// TIA Portal V20 export
FUNCTION "SafetyState" : Void   // FC97, LAD
// stored: SetENOAutomatically false
   VAR CONSTANT
      TRUE : Bool := TRUE;
      FALSE : Bool;
   END_VAR
   VAR_TEMP   // added for the SCL form of the ladder/FBD networks
      _w1 : Bool;
   END_VAR
BEGIN

REGION Network 1: Stack Door Common Monitoring#1
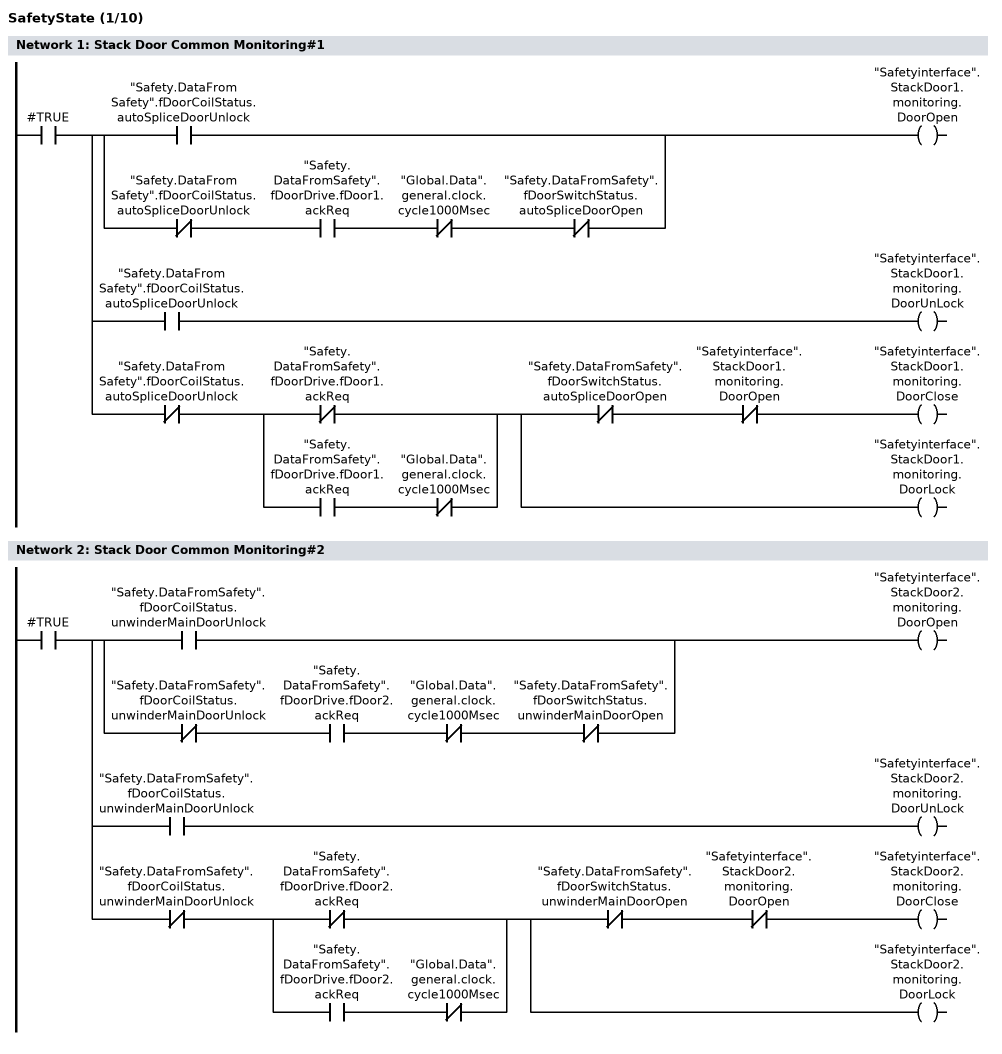
   RUNG wire#powerrail
      Contact( #TRUE )
      wire#w1
      Contact( "Safety.DataFromSafety".fDoorCoilStatus.autoSpliceDoorUnlock )
      wire#w2
      Coil( "Safetyinterface".StackDoor1.monitoring.DoorOpen )
   END_RUNG
   RUNG wire#w1
      I_Contact( "Safety.DataFromSafety".fDoorCoilStatus.autoSpliceDoorUnlock )
      Contact( "Safety.DataFromSafety".fDoorDrive.fDoor1.ackReq )
      I_Contact( "Global.Data".general.clock.cycle1000Msec )
      I_Contact( "Safety.DataFromSafety".fDoorSwitchStatus.autoSpliceDoorOpen )
   END_RUNG wire#w2
   RUNG wire#w1
      Contact( "Safety.DataFromSafety".fDoorCoilStatus.autoSpliceDoorUnlock )
      Coil( "Safetyinterface".StackDoor1.monitoring.DoorUnLock )
   END_RUNG
   RUNG wire#w1
      I_Contact( "Safety.DataFromSafety".fDoorCoilStatus.autoSpliceDoorUnlock )
      wire#w3
      I_Contact( "Safety.DataFromSafety".fDoorDrive.fDoor1.ackReq )
      wire#w4
      I_Contact( "Safety.DataFromSafety".fDoorSwitchStatus.autoSpliceDoorOpen )
      I_Contact( "Safetyinterface".StackDoor1.monitoring.DoorOpen )
      Coil( "Safetyinterface".StackDoor1.monitoring.DoorClose )
   END_RUNG
   RUNG wire#w3
      Contact( "Safety.DataFromSafety".fDoorDrive.fDoor1.ackReq )
      I_Contact( "Global.Data".general.clock.cycle1000Msec )
   END_RUNG wire#w4
   RUNG wire#w4
      Coil( "Safetyinterface".StackDoor1.monitoring.DoorLock )
   END_RUNG
   // the same network as SCL:
   "Safetyinterface".StackDoor1.monitoring.DoorOpen := #TRUE AND ("Safety.DataFromSafety".fDoorCoilStatus.autoSpliceDoorUnlock OR (NOT "Safety.DataFromSafety".fDoorCoilStatus.autoSpliceDoorUnlock AND "Safety.DataFromSafety".fDoorDrive.fDoor1.ackReq AND NOT "Global.Data".general.clock.cycle1000Msec AND NOT "Safety.DataFromSafety".fDoorSwitchStatus.autoSpliceDoorOpen));
   "Safetyinterface".StackDoor1.monitoring.DoorUnLock := #TRUE AND "Safety.DataFromSafety".fDoorCoilStatus.autoSpliceDoorUnlock;
   #_w1 := #TRUE AND NOT "Safety.DataFromSafety".fDoorCoilStatus.autoSpliceDoorUnlock AND (NOT "Safety.DataFromSafety".fDoorDrive.fDoor1.ackReq OR ("Safety.DataFromSafety".fDoorDrive.fDoor1.ackReq AND NOT "Global.Data".general.clock.cycle1000Msec));
   "Safetyinterface".StackDoor1.monitoring.DoorClose := #_w1 AND NOT "Safety.DataFromSafety".fDoorSwitchStatus.autoSpliceDoorOpen AND NOT "Safetyinterface".StackDoor1.monitoring.DoorOpen;
   "Safetyinterface".StackDoor1.monitoring.DoorLock := #_w1;
END_REGION

REGION Network 2: Stack Door Common Monitoring#2
   RUNG wire#powerrail
      Contact( #TRUE )
      wire#w1
      Contact( "Safety.DataFromSafety".fDoorCoilStatus.unwinderMainDoorUnlock )
      wire#w2
      Coil( "Safetyinterface".StackDoor2.monitoring.DoorOpen )
   END_RUNG
   RUNG wire#w1
      I_Contact( "Safety.DataFromSafety".fDoorCoilStatus.unwinderMainDoorUnlock )
      Contact( "Safety.DataFromSafety".fDoorDrive.fDoor2.ackReq )
      I_Contact( "Global.Data".general.clock.cycle1000Msec )
      I_Contact( "Safety.DataFromSafety".fDoorSwitchStatus.unwinderMainDoorOpen )
   END_RUNG wire#w2
   RUNG wire#w1
      Contact( "Safety.DataFromSafety".fDoorCoilStatus.unwinderMainDoorUnlock )
      Coil( "Safetyinterface".StackDoor2.monitoring.DoorUnLock )
   END_RUNG
   RUNG wire#w1
      I_Contact( "Safety.DataFromSafety".fDoorCoilStatus.unwinderMainDoorUnlock )
      wire#w3
      I_Contact( "Safety.DataFromSafety".fDoorDrive.fDoor2.ackReq )
      wire#w4
      I_Contact( "Safety.DataFromSafety".fDoorSwitchStatus.unwinderMainDoorOpen )
      I_Contact( "Safetyinterface".StackDoor2.monitoring.DoorOpen )
      Coil( "Safetyinterface".StackDoor2.monitoring.DoorClose )
   END_RUNG
   RUNG wire#w3
      Contact( "Safety.DataFromSafety".fDoorDrive.fDoor2.ackReq )
      I_Contact( "Global.Data".general.clock.cycle1000Msec )
   END_RUNG wire#w4
   RUNG wire#w4
      Coil( "Safetyinterface".StackDoor2.monitoring.DoorLock )
   END_RUNG
   // the same network as SCL:
   "Safetyinterface".StackDoor2.monitoring.DoorOpen := #TRUE AND ("Safety.DataFromSafety".fDoorCoilStatus.unwinderMainDoorUnlock OR (NOT "Safety.DataFromSafety".fDoorCoilStatus.unwinderMainDoorUnlock AND "Safety.DataFromSafety".fDoorDrive.fDoor2.ackReq AND NOT "Global.Data".general.clock.cycle1000Msec AND NOT "Safety.DataFromSafety".fDoorSwitchStatus.unwinderMainDoorOpen));
   "Safetyinterface".StackDoor2.monitoring.DoorUnLock := #TRUE AND "Safety.DataFromSafety".fDoorCoilStatus.unwinderMainDoorUnlock;
   #_w1 := #TRUE AND NOT "Safety.DataFromSafety".fDoorCoilStatus.unwinderMainDoorUnlock AND (NOT "Safety.DataFromSafety".fDoorDrive.fDoor2.ackReq OR ("Safety.DataFromSafety".fDoorDrive.fDoor2.ackReq AND NOT "Global.Data".general.clock.cycle1000Msec));
   "Safetyinterface".StackDoor2.monitoring.DoorClose := #_w1 AND NOT "Safety.DataFromSafety".fDoorSwitchStatus.unwinderMainDoorOpen AND NOT "Safetyinterface".StackDoor2.monitoring.DoorOpen;
   "Safetyinterface".StackDoor2.monitoring.DoorLock := #_w1;
END_REGION

REGION Network 3: Stack Door Common Monitoring#3
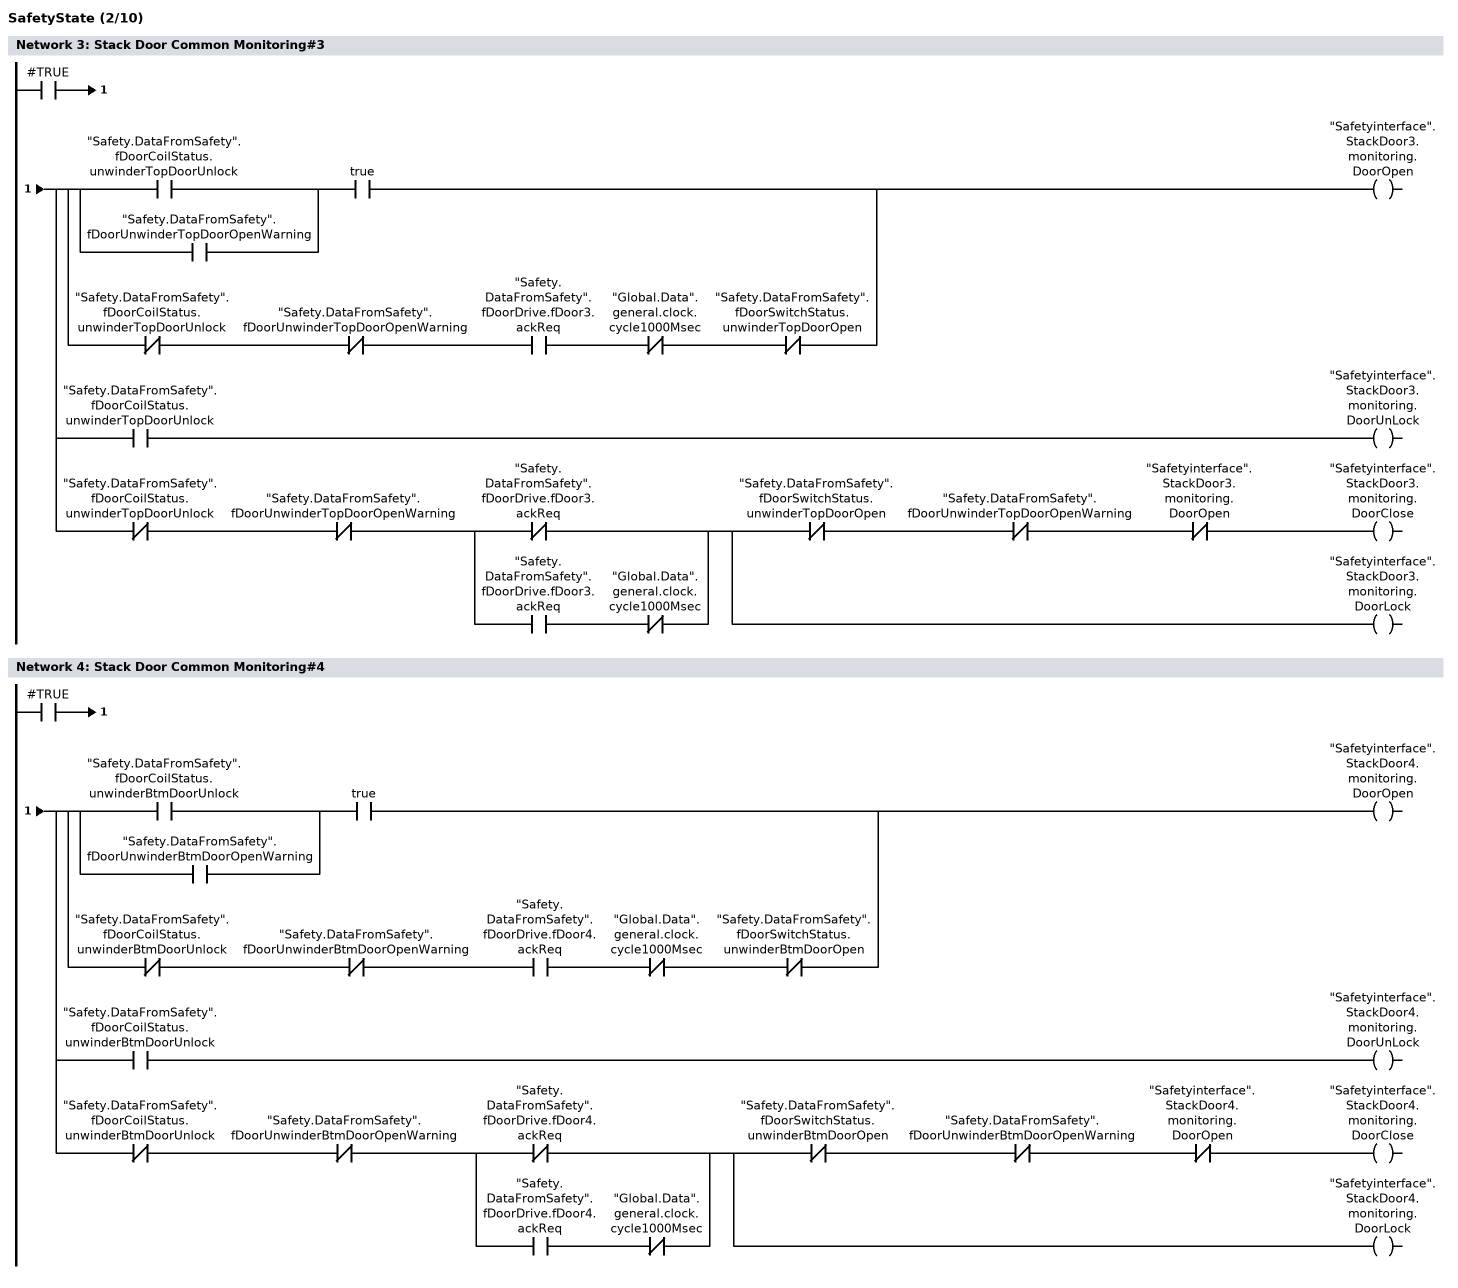
   RUNG wire#powerrail
      Contact( #TRUE )
      wire#w1
      Contact( "Safety.DataFromSafety".fDoorCoilStatus.unwinderTopDoorUnlock )
      wire#w2
      Contact( true )
      wire#w3
      Coil( "Safetyinterface".StackDoor3.monitoring.DoorOpen )
   END_RUNG
   RUNG wire#w1
      Contact( "Safety.DataFromSafety".fDoorUnwinderTopDoorOpenWarning )
   END_RUNG wire#w2
   RUNG wire#w1
      I_Contact( "Safety.DataFromSafety".fDoorCoilStatus.unwinderTopDoorUnlock )
      I_Contact( "Safety.DataFromSafety".fDoorUnwinderTopDoorOpenWarning )
      Contact( "Safety.DataFromSafety".fDoorDrive.fDoor3.ackReq )
      I_Contact( "Global.Data".general.clock.cycle1000Msec )
      I_Contact( "Safety.DataFromSafety".fDoorSwitchStatus.unwinderTopDoorOpen )
   END_RUNG wire#w3
   RUNG wire#w1
      Contact( "Safety.DataFromSafety".fDoorCoilStatus.unwinderTopDoorUnlock )
      Coil( "Safetyinterface".StackDoor3.monitoring.DoorUnLock )
   END_RUNG
   RUNG wire#w1
      I_Contact( "Safety.DataFromSafety".fDoorCoilStatus.unwinderTopDoorUnlock )
      I_Contact( "Safety.DataFromSafety".fDoorUnwinderTopDoorOpenWarning )
      wire#w4
      I_Contact( "Safety.DataFromSafety".fDoorDrive.fDoor3.ackReq )
      wire#w5
      I_Contact( "Safety.DataFromSafety".fDoorSwitchStatus.unwinderTopDoorOpen )
      I_Contact( "Safety.DataFromSafety".fDoorUnwinderTopDoorOpenWarning )
      I_Contact( "Safetyinterface".StackDoor3.monitoring.DoorOpen )
      Coil( "Safetyinterface".StackDoor3.monitoring.DoorClose )
   END_RUNG
   RUNG wire#w4
      Contact( "Safety.DataFromSafety".fDoorDrive.fDoor3.ackReq )
      I_Contact( "Global.Data".general.clock.cycle1000Msec )
   END_RUNG wire#w5
   RUNG wire#w5
      Coil( "Safetyinterface".StackDoor3.monitoring.DoorLock )
   END_RUNG
   // the same network as SCL:
   "Safetyinterface".StackDoor3.monitoring.DoorOpen := #TRUE AND ((("Safety.DataFromSafety".fDoorCoilStatus.unwinderTopDoorUnlock OR "Safety.DataFromSafety".fDoorUnwinderTopDoorOpenWarning) AND true) OR (NOT "Safety.DataFromSafety".fDoorCoilStatus.unwinderTopDoorUnlock AND NOT "Safety.DataFromSafety".fDoorUnwinderTopDoorOpenWarning AND "Safety.DataFromSafety".fDoorDrive.fDoor3.ackReq AND NOT "Global.Data".general.clock.cycle1000Msec AND NOT "Safety.DataFromSafety".fDoorSwitchStatus.unwinderTopDoorOpen));
   "Safetyinterface".StackDoor3.monitoring.DoorUnLock := #TRUE AND "Safety.DataFromSafety".fDoorCoilStatus.unwinderTopDoorUnlock;
   #_w1 := #TRUE AND NOT "Safety.DataFromSafety".fDoorCoilStatus.unwinderTopDoorUnlock AND NOT "Safety.DataFromSafety".fDoorUnwinderTopDoorOpenWarning AND (NOT "Safety.DataFromSafety".fDoorDrive.fDoor3.ackReq OR ("Safety.DataFromSafety".fDoorDrive.fDoor3.ackReq AND NOT "Global.Data".general.clock.cycle1000Msec));
   "Safetyinterface".StackDoor3.monitoring.DoorClose := #_w1 AND NOT "Safety.DataFromSafety".fDoorSwitchStatus.unwinderTopDoorOpen AND NOT "Safety.DataFromSafety".fDoorUnwinderTopDoorOpenWarning AND NOT "Safetyinterface".StackDoor3.monitoring.DoorOpen;
   "Safetyinterface".StackDoor3.monitoring.DoorLock := #_w1;
END_REGION

REGION Network 4: Stack Door Common Monitoring#4
   RUNG wire#powerrail
      Contact( #TRUE )
      wire#w1
      Contact( "Safety.DataFromSafety".fDoorCoilStatus.unwinderBtmDoorUnlock )
      wire#w2
      Contact( true )
      wire#w3
      Coil( "Safetyinterface".StackDoor4.monitoring.DoorOpen )
   END_RUNG
   RUNG wire#w1
      Contact( "Safety.DataFromSafety".fDoorUnwinderBtmDoorOpenWarning )
   END_RUNG wire#w2
   RUNG wire#w1
      I_Contact( "Safety.DataFromSafety".fDoorCoilStatus.unwinderBtmDoorUnlock )
      I_Contact( "Safety.DataFromSafety".fDoorUnwinderBtmDoorOpenWarning )
      Contact( "Safety.DataFromSafety".fDoorDrive.fDoor4.ackReq )
      I_Contact( "Global.Data".general.clock.cycle1000Msec )
      I_Contact( "Safety.DataFromSafety".fDoorSwitchStatus.unwinderBtmDoorOpen )
   END_RUNG wire#w3
   RUNG wire#w1
      Contact( "Safety.DataFromSafety".fDoorCoilStatus.unwinderBtmDoorUnlock )
      Coil( "Safetyinterface".StackDoor4.monitoring.DoorUnLock )
   END_RUNG
   RUNG wire#w1
      I_Contact( "Safety.DataFromSafety".fDoorCoilStatus.unwinderBtmDoorUnlock )
      I_Contact( "Safety.DataFromSafety".fDoorUnwinderBtmDoorOpenWarning )
      wire#w4
      I_Contact( "Safety.DataFromSafety".fDoorDrive.fDoor4.ackReq )
      wire#w5
      I_Contact( "Safety.DataFromSafety".fDoorSwitchStatus.unwinderBtmDoorOpen )
      I_Contact( "Safety.DataFromSafety".fDoorUnwinderBtmDoorOpenWarning )
      I_Contact( "Safetyinterface".StackDoor4.monitoring.DoorOpen )
      Coil( "Safetyinterface".StackDoor4.monitoring.DoorClose )
   END_RUNG
   RUNG wire#w4
      Contact( "Safety.DataFromSafety".fDoorDrive.fDoor4.ackReq )
      I_Contact( "Global.Data".general.clock.cycle1000Msec )
   END_RUNG wire#w5
   RUNG wire#w5
      Coil( "Safetyinterface".StackDoor4.monitoring.DoorLock )
   END_RUNG
   // the same network as SCL:
   "Safetyinterface".StackDoor4.monitoring.DoorOpen := #TRUE AND ((("Safety.DataFromSafety".fDoorCoilStatus.unwinderBtmDoorUnlock OR "Safety.DataFromSafety".fDoorUnwinderBtmDoorOpenWarning) AND true) OR (NOT "Safety.DataFromSafety".fDoorCoilStatus.unwinderBtmDoorUnlock AND NOT "Safety.DataFromSafety".fDoorUnwinderBtmDoorOpenWarning AND "Safety.DataFromSafety".fDoorDrive.fDoor4.ackReq AND NOT "Global.Data".general.clock.cycle1000Msec AND NOT "Safety.DataFromSafety".fDoorSwitchStatus.unwinderBtmDoorOpen));
   "Safetyinterface".StackDoor4.monitoring.DoorUnLock := #TRUE AND "Safety.DataFromSafety".fDoorCoilStatus.unwinderBtmDoorUnlock;
   #_w1 := #TRUE AND NOT "Safety.DataFromSafety".fDoorCoilStatus.unwinderBtmDoorUnlock AND NOT "Safety.DataFromSafety".fDoorUnwinderBtmDoorOpenWarning AND (NOT "Safety.DataFromSafety".fDoorDrive.fDoor4.ackReq OR ("Safety.DataFromSafety".fDoorDrive.fDoor4.ackReq AND NOT "Global.Data".general.clock.cycle1000Msec));
   "Safetyinterface".StackDoor4.monitoring.DoorClose := #_w1 AND NOT "Safety.DataFromSafety".fDoorSwitchStatus.unwinderBtmDoorOpen AND NOT "Safety.DataFromSafety".fDoorUnwinderBtmDoorOpenWarning AND NOT "Safetyinterface".StackDoor4.monitoring.DoorOpen;
   "Safetyinterface".StackDoor4.monitoring.DoorLock := #_w1;
END_REGION

REGION Network 5: Stack Door Common Command#5
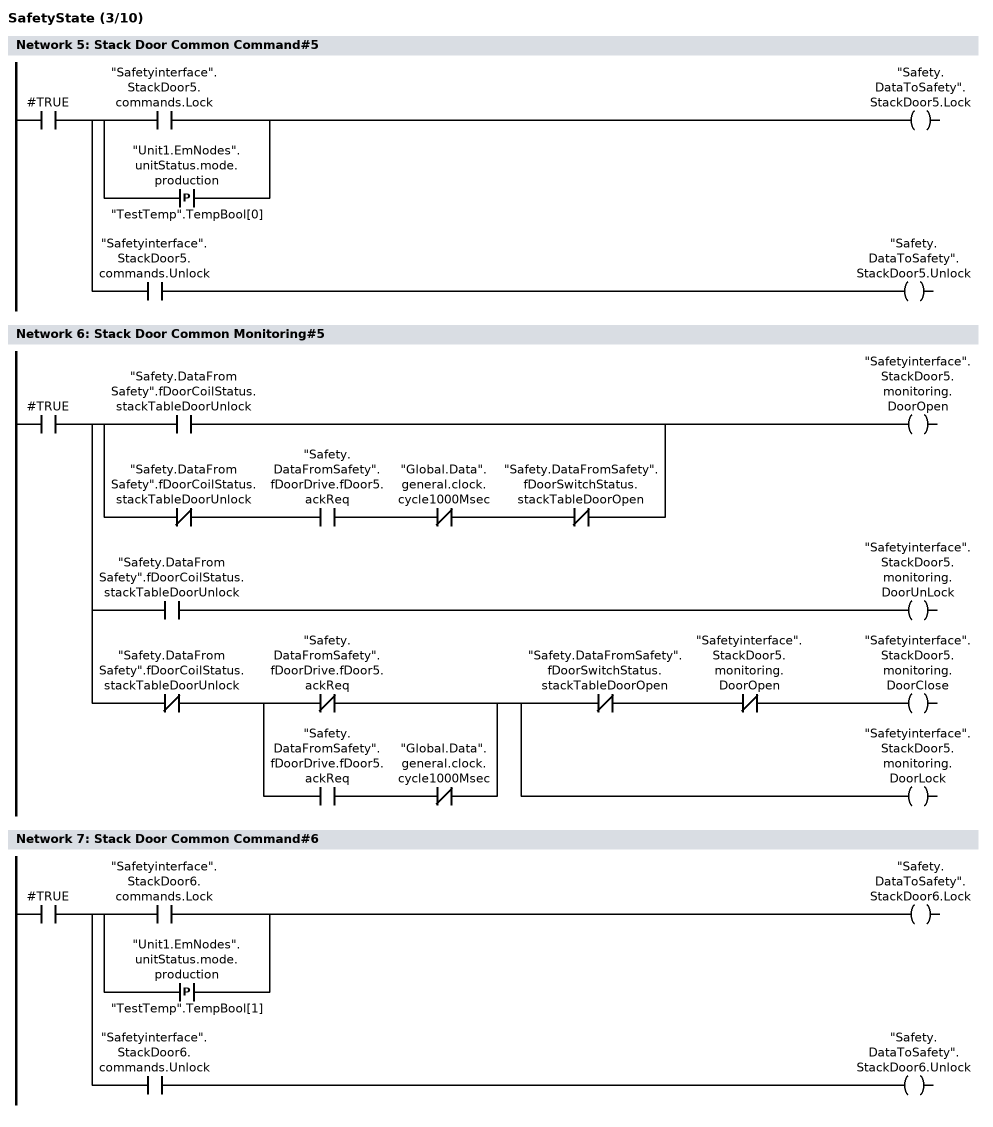
   RUNG wire#powerrail
      Contact( #TRUE )
      wire#w1
      Contact( "Safetyinterface".StackDoor5.commands.Lock )
      wire#w2
      Coil( "Safety.DataToSafety".StackDoor5.Lock )
   END_RUNG
   RUNG wire#w1
      P_Contact(operand := "Unit1.EmNodes".unitStatus.mode.production, bit := "TestTemp".TempBool[0])
   END_RUNG wire#w2
   RUNG wire#w1
      Contact( "Safetyinterface".StackDoor5.commands.Unlock )
      Coil( "Safety.DataToSafety".StackDoor5.Unlock )
   END_RUNG
   // the same network as SCL:
   #_w1 := #TRUE AND "Unit1.EmNodes".unitStatus.mode.production AND NOT "TestTemp".TempBool[0];   // rising edge of "Unit1.EmNodes".unitStatus.mode.production
   "TestTemp".TempBool[0] := "Unit1.EmNodes".unitStatus.mode.production;
   "Safety.DataToSafety".StackDoor5.Lock := (#TRUE AND "Safetyinterface".StackDoor5.commands.Lock) OR #_w1;
   "Safety.DataToSafety".StackDoor5.Unlock := #TRUE AND "Safetyinterface".StackDoor5.commands.Unlock;
END_REGION

REGION Network 6: Stack Door Common Monitoring#5
   RUNG wire#powerrail
      Contact( #TRUE )
      wire#w1
      Contact( "Safety.DataFromSafety".fDoorCoilStatus.stackTableDoorUnlock )
      wire#w2
      Coil( "Safetyinterface".StackDoor5.monitoring.DoorOpen )
   END_RUNG
   RUNG wire#w1
      I_Contact( "Safety.DataFromSafety".fDoorCoilStatus.stackTableDoorUnlock )
      Contact( "Safety.DataFromSafety".fDoorDrive.fDoor5.ackReq )
      I_Contact( "Global.Data".general.clock.cycle1000Msec )
      I_Contact( "Safety.DataFromSafety".fDoorSwitchStatus.stackTableDoorOpen )
   END_RUNG wire#w2
   RUNG wire#w1
      Contact( "Safety.DataFromSafety".fDoorCoilStatus.stackTableDoorUnlock )
      Coil( "Safetyinterface".StackDoor5.monitoring.DoorUnLock )
   END_RUNG
   RUNG wire#w1
      I_Contact( "Safety.DataFromSafety".fDoorCoilStatus.stackTableDoorUnlock )
      wire#w3
      I_Contact( "Safety.DataFromSafety".fDoorDrive.fDoor5.ackReq )
      wire#w4
      I_Contact( "Safety.DataFromSafety".fDoorSwitchStatus.stackTableDoorOpen )
      I_Contact( "Safetyinterface".StackDoor5.monitoring.DoorOpen )
      Coil( "Safetyinterface".StackDoor5.monitoring.DoorClose )
   END_RUNG
   RUNG wire#w3
      Contact( "Safety.DataFromSafety".fDoorDrive.fDoor5.ackReq )
      I_Contact( "Global.Data".general.clock.cycle1000Msec )
   END_RUNG wire#w4
   RUNG wire#w4
      Coil( "Safetyinterface".StackDoor5.monitoring.DoorLock )
   END_RUNG
   // the same network as SCL:
   "Safetyinterface".StackDoor5.monitoring.DoorOpen := #TRUE AND ("Safety.DataFromSafety".fDoorCoilStatus.stackTableDoorUnlock OR (NOT "Safety.DataFromSafety".fDoorCoilStatus.stackTableDoorUnlock AND "Safety.DataFromSafety".fDoorDrive.fDoor5.ackReq AND NOT "Global.Data".general.clock.cycle1000Msec AND NOT "Safety.DataFromSafety".fDoorSwitchStatus.stackTableDoorOpen));
   "Safetyinterface".StackDoor5.monitoring.DoorUnLock := #TRUE AND "Safety.DataFromSafety".fDoorCoilStatus.stackTableDoorUnlock;
   #_w1 := #TRUE AND NOT "Safety.DataFromSafety".fDoorCoilStatus.stackTableDoorUnlock AND (NOT "Safety.DataFromSafety".fDoorDrive.fDoor5.ackReq OR ("Safety.DataFromSafety".fDoorDrive.fDoor5.ackReq AND NOT "Global.Data".general.clock.cycle1000Msec));
   "Safetyinterface".StackDoor5.monitoring.DoorClose := #_w1 AND NOT "Safety.DataFromSafety".fDoorSwitchStatus.stackTableDoorOpen AND NOT "Safetyinterface".StackDoor5.monitoring.DoorOpen;
   "Safetyinterface".StackDoor5.monitoring.DoorLock := #_w1;
END_REGION

REGION Network 7: Stack Door Common Command#6
   RUNG wire#powerrail
      Contact( #TRUE )
      wire#w1
      Contact( "Safetyinterface".StackDoor6.commands.Lock )
      wire#w2
      Coil( "Safety.DataToSafety".StackDoor6.Lock )
   END_RUNG
   RUNG wire#w1
      P_Contact(operand := "Unit1.EmNodes".unitStatus.mode.production, bit := "TestTemp".TempBool[1])
   END_RUNG wire#w2
   RUNG wire#w1
      Contact( "Safetyinterface".StackDoor6.commands.Unlock )
      Coil( "Safety.DataToSafety".StackDoor6.Unlock )
   END_RUNG
   // the same network as SCL:
   #_w1 := #TRUE AND "Unit1.EmNodes".unitStatus.mode.production AND NOT "TestTemp".TempBool[1];   // rising edge of "Unit1.EmNodes".unitStatus.mode.production
   "TestTemp".TempBool[1] := "Unit1.EmNodes".unitStatus.mode.production;
   "Safety.DataToSafety".StackDoor6.Lock := (#TRUE AND "Safetyinterface".StackDoor6.commands.Lock) OR #_w1;
   "Safety.DataToSafety".StackDoor6.Unlock := #TRUE AND "Safetyinterface".StackDoor6.commands.Unlock;
END_REGION

REGION Network 8: Stack Door Common Monitoring#6
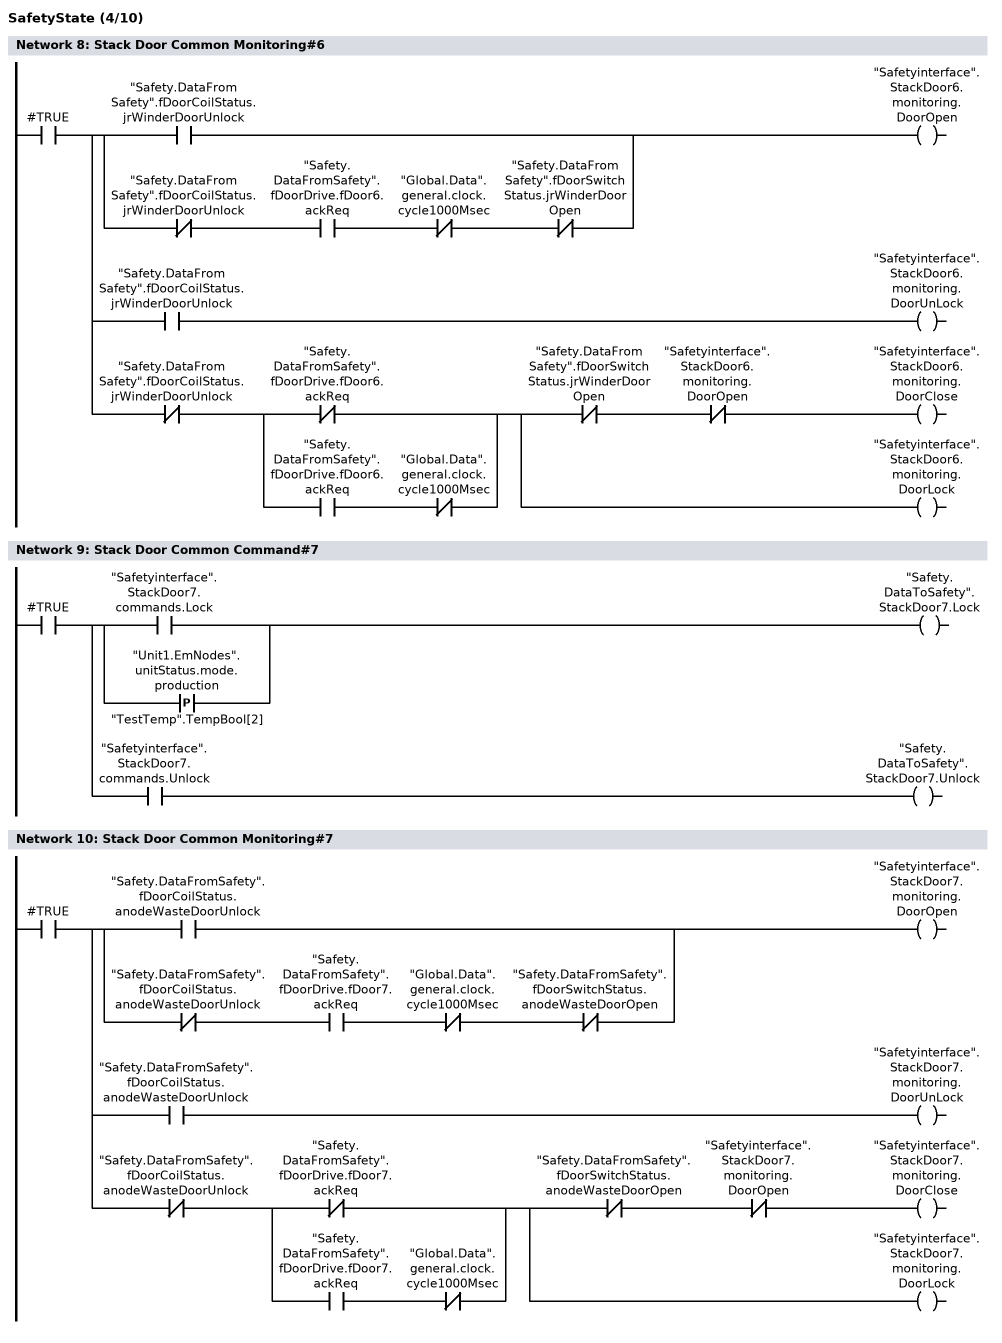
   RUNG wire#powerrail
      Contact( #TRUE )
      wire#w1
      Contact( "Safety.DataFromSafety".fDoorCoilStatus.jrWinderDoorUnlock )
      wire#w2
      Coil( "Safetyinterface".StackDoor6.monitoring.DoorOpen )
   END_RUNG
   RUNG wire#w1
      I_Contact( "Safety.DataFromSafety".fDoorCoilStatus.jrWinderDoorUnlock )
      Contact( "Safety.DataFromSafety".fDoorDrive.fDoor6.ackReq )
      I_Contact( "Global.Data".general.clock.cycle1000Msec )
      I_Contact( "Safety.DataFromSafety".fDoorSwitchStatus.jrWinderDoorOpen )
   END_RUNG wire#w2
   RUNG wire#w1
      Contact( "Safety.DataFromSafety".fDoorCoilStatus.jrWinderDoorUnlock )
      Coil( "Safetyinterface".StackDoor6.monitoring.DoorUnLock )
   END_RUNG
   RUNG wire#w1
      I_Contact( "Safety.DataFromSafety".fDoorCoilStatus.jrWinderDoorUnlock )
      wire#w3
      I_Contact( "Safety.DataFromSafety".fDoorDrive.fDoor6.ackReq )
      wire#w4
      I_Contact( "Safety.DataFromSafety".fDoorSwitchStatus.jrWinderDoorOpen )
      I_Contact( "Safetyinterface".StackDoor6.monitoring.DoorOpen )
      Coil( "Safetyinterface".StackDoor6.monitoring.DoorClose )
   END_RUNG
   RUNG wire#w3
      Contact( "Safety.DataFromSafety".fDoorDrive.fDoor6.ackReq )
      I_Contact( "Global.Data".general.clock.cycle1000Msec )
   END_RUNG wire#w4
   RUNG wire#w4
      Coil( "Safetyinterface".StackDoor6.monitoring.DoorLock )
   END_RUNG
   // the same network as SCL:
   "Safetyinterface".StackDoor6.monitoring.DoorOpen := #TRUE AND ("Safety.DataFromSafety".fDoorCoilStatus.jrWinderDoorUnlock OR (NOT "Safety.DataFromSafety".fDoorCoilStatus.jrWinderDoorUnlock AND "Safety.DataFromSafety".fDoorDrive.fDoor6.ackReq AND NOT "Global.Data".general.clock.cycle1000Msec AND NOT "Safety.DataFromSafety".fDoorSwitchStatus.jrWinderDoorOpen));
   "Safetyinterface".StackDoor6.monitoring.DoorUnLock := #TRUE AND "Safety.DataFromSafety".fDoorCoilStatus.jrWinderDoorUnlock;
   #_w1 := #TRUE AND NOT "Safety.DataFromSafety".fDoorCoilStatus.jrWinderDoorUnlock AND (NOT "Safety.DataFromSafety".fDoorDrive.fDoor6.ackReq OR ("Safety.DataFromSafety".fDoorDrive.fDoor6.ackReq AND NOT "Global.Data".general.clock.cycle1000Msec));
   "Safetyinterface".StackDoor6.monitoring.DoorClose := #_w1 AND NOT "Safety.DataFromSafety".fDoorSwitchStatus.jrWinderDoorOpen AND NOT "Safetyinterface".StackDoor6.monitoring.DoorOpen;
   "Safetyinterface".StackDoor6.monitoring.DoorLock := #_w1;
END_REGION

REGION Network 9: Stack Door Common Command#7
   RUNG wire#powerrail
      Contact( #TRUE )
      wire#w1
      Contact( "Safetyinterface".StackDoor7.commands.Lock )
      wire#w2
      Coil( "Safety.DataToSafety".StackDoor7.Lock )
   END_RUNG
   RUNG wire#w1
      P_Contact(operand := "Unit1.EmNodes".unitStatus.mode.production, bit := "TestTemp".TempBool[2])
   END_RUNG wire#w2
   RUNG wire#w1
      Contact( "Safetyinterface".StackDoor7.commands.Unlock )
      Coil( "Safety.DataToSafety".StackDoor7.Unlock )
   END_RUNG
   // the same network as SCL:
   #_w1 := #TRUE AND "Unit1.EmNodes".unitStatus.mode.production AND NOT "TestTemp".TempBool[2];   // rising edge of "Unit1.EmNodes".unitStatus.mode.production
   "TestTemp".TempBool[2] := "Unit1.EmNodes".unitStatus.mode.production;
   "Safety.DataToSafety".StackDoor7.Lock := (#TRUE AND "Safetyinterface".StackDoor7.commands.Lock) OR #_w1;
   "Safety.DataToSafety".StackDoor7.Unlock := #TRUE AND "Safetyinterface".StackDoor7.commands.Unlock;
END_REGION

REGION Network 10: Stack Door Common Monitoring#7
   RUNG wire#powerrail
      Contact( #TRUE )
      wire#w1
      Contact( "Safety.DataFromSafety".fDoorCoilStatus.anodeWasteDoorUnlock )
      wire#w2
      Coil( "Safetyinterface".StackDoor7.monitoring.DoorOpen )
   END_RUNG
   RUNG wire#w1
      I_Contact( "Safety.DataFromSafety".fDoorCoilStatus.anodeWasteDoorUnlock )
      Contact( "Safety.DataFromSafety".fDoorDrive.fDoor7.ackReq )
      I_Contact( "Global.Data".general.clock.cycle1000Msec )
      I_Contact( "Safety.DataFromSafety".fDoorSwitchStatus.anodeWasteDoorOpen )
   END_RUNG wire#w2
   RUNG wire#w1
      Contact( "Safety.DataFromSafety".fDoorCoilStatus.anodeWasteDoorUnlock )
      Coil( "Safetyinterface".StackDoor7.monitoring.DoorUnLock )
   END_RUNG
   RUNG wire#w1
      I_Contact( "Safety.DataFromSafety".fDoorCoilStatus.anodeWasteDoorUnlock )
      wire#w3
      I_Contact( "Safety.DataFromSafety".fDoorDrive.fDoor7.ackReq )
      wire#w4
      I_Contact( "Safety.DataFromSafety".fDoorSwitchStatus.anodeWasteDoorOpen )
      I_Contact( "Safetyinterface".StackDoor7.monitoring.DoorOpen )
      Coil( "Safetyinterface".StackDoor7.monitoring.DoorClose )
   END_RUNG
   RUNG wire#w3
      Contact( "Safety.DataFromSafety".fDoorDrive.fDoor7.ackReq )
      I_Contact( "Global.Data".general.clock.cycle1000Msec )
   END_RUNG wire#w4
   RUNG wire#w4
      Coil( "Safetyinterface".StackDoor7.monitoring.DoorLock )
   END_RUNG
   // the same network as SCL:
   "Safetyinterface".StackDoor7.monitoring.DoorOpen := #TRUE AND ("Safety.DataFromSafety".fDoorCoilStatus.anodeWasteDoorUnlock OR (NOT "Safety.DataFromSafety".fDoorCoilStatus.anodeWasteDoorUnlock AND "Safety.DataFromSafety".fDoorDrive.fDoor7.ackReq AND NOT "Global.Data".general.clock.cycle1000Msec AND NOT "Safety.DataFromSafety".fDoorSwitchStatus.anodeWasteDoorOpen));
   "Safetyinterface".StackDoor7.monitoring.DoorUnLock := #TRUE AND "Safety.DataFromSafety".fDoorCoilStatus.anodeWasteDoorUnlock;
   #_w1 := #TRUE AND NOT "Safety.DataFromSafety".fDoorCoilStatus.anodeWasteDoorUnlock AND (NOT "Safety.DataFromSafety".fDoorDrive.fDoor7.ackReq OR ("Safety.DataFromSafety".fDoorDrive.fDoor7.ackReq AND NOT "Global.Data".general.clock.cycle1000Msec));
   "Safetyinterface".StackDoor7.monitoring.DoorClose := #_w1 AND NOT "Safety.DataFromSafety".fDoorSwitchStatus.anodeWasteDoorOpen AND NOT "Safetyinterface".StackDoor7.monitoring.DoorOpen;
   "Safetyinterface".StackDoor7.monitoring.DoorLock := #_w1;
END_REGION

REGION Network 11: Stack Door Common Command#8
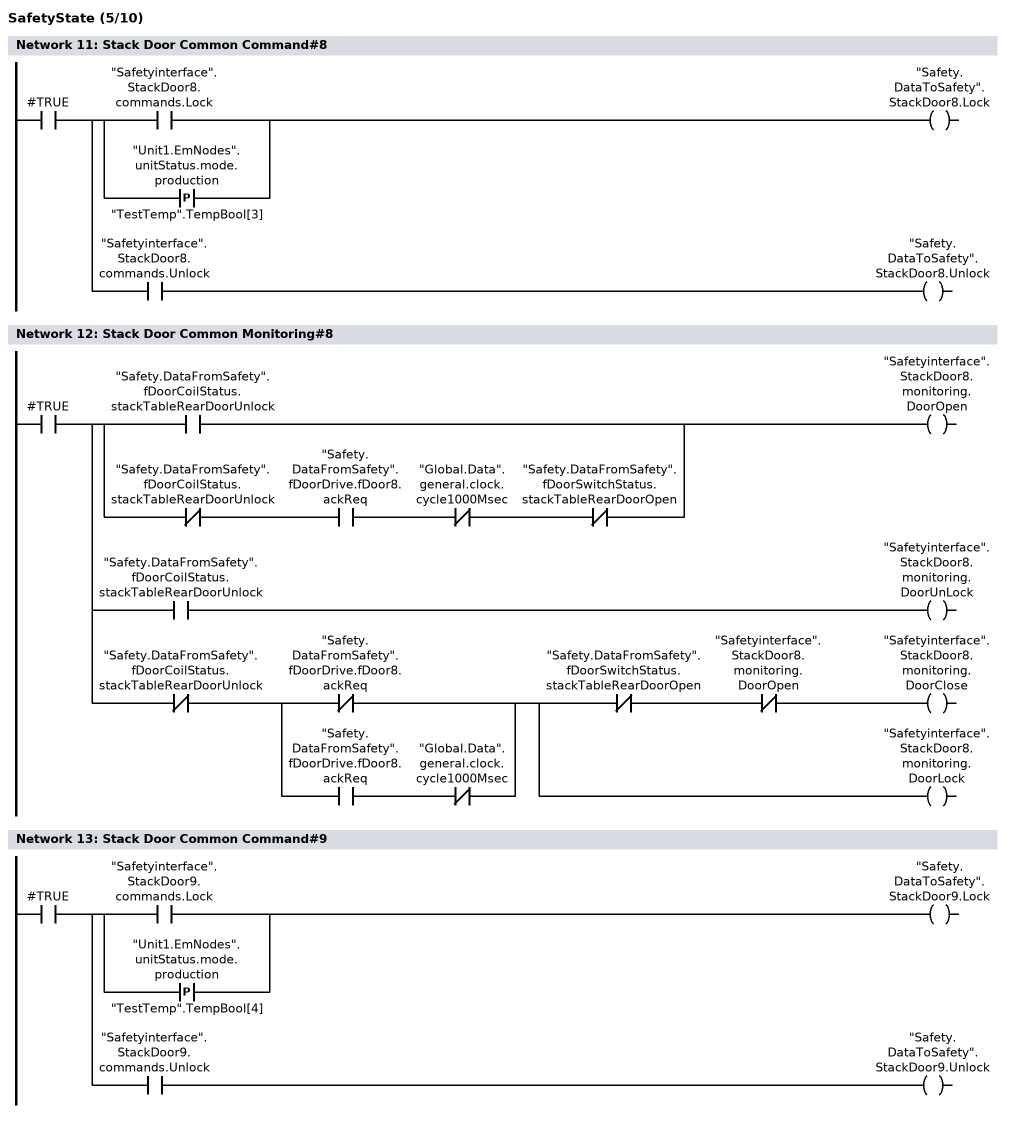
   RUNG wire#powerrail
      Contact( #TRUE )
      wire#w1
      Contact( "Safetyinterface".StackDoor8.commands.Lock )
      wire#w2
      Coil( "Safety.DataToSafety".StackDoor8.Lock )
   END_RUNG
   RUNG wire#w1
      P_Contact(operand := "Unit1.EmNodes".unitStatus.mode.production, bit := "TestTemp".TempBool[3])
   END_RUNG wire#w2
   RUNG wire#w1
      Contact( "Safetyinterface".StackDoor8.commands.Unlock )
      Coil( "Safety.DataToSafety".StackDoor8.Unlock )
   END_RUNG
   // the same network as SCL:
   #_w1 := #TRUE AND "Unit1.EmNodes".unitStatus.mode.production AND NOT "TestTemp".TempBool[3];   // rising edge of "Unit1.EmNodes".unitStatus.mode.production
   "TestTemp".TempBool[3] := "Unit1.EmNodes".unitStatus.mode.production;
   "Safety.DataToSafety".StackDoor8.Lock := (#TRUE AND "Safetyinterface".StackDoor8.commands.Lock) OR #_w1;
   "Safety.DataToSafety".StackDoor8.Unlock := #TRUE AND "Safetyinterface".StackDoor8.commands.Unlock;
END_REGION

REGION Network 12: Stack Door Common Monitoring#8
   RUNG wire#powerrail
      Contact( #TRUE )
      wire#w1
      Contact( "Safety.DataFromSafety".fDoorCoilStatus.stackTableRearDoorUnlock )
      wire#w2
      Coil( "Safetyinterface".StackDoor8.monitoring.DoorOpen )
   END_RUNG
   RUNG wire#w1
      I_Contact( "Safety.DataFromSafety".fDoorCoilStatus.stackTableRearDoorUnlock )
      Contact( "Safety.DataFromSafety".fDoorDrive.fDoor8.ackReq )
      I_Contact( "Global.Data".general.clock.cycle1000Msec )
      I_Contact( "Safety.DataFromSafety".fDoorSwitchStatus.stackTableRearDoorOpen )
   END_RUNG wire#w2
   RUNG wire#w1
      Contact( "Safety.DataFromSafety".fDoorCoilStatus.stackTableRearDoorUnlock )
      Coil( "Safetyinterface".StackDoor8.monitoring.DoorUnLock )
   END_RUNG
   RUNG wire#w1
      I_Contact( "Safety.DataFromSafety".fDoorCoilStatus.stackTableRearDoorUnlock )
      wire#w3
      I_Contact( "Safety.DataFromSafety".fDoorDrive.fDoor8.ackReq )
      wire#w4
      I_Contact( "Safety.DataFromSafety".fDoorSwitchStatus.stackTableRearDoorOpen )
      I_Contact( "Safetyinterface".StackDoor8.monitoring.DoorOpen )
      Coil( "Safetyinterface".StackDoor8.monitoring.DoorClose )
   END_RUNG
   RUNG wire#w3
      Contact( "Safety.DataFromSafety".fDoorDrive.fDoor8.ackReq )
      I_Contact( "Global.Data".general.clock.cycle1000Msec )
   END_RUNG wire#w4
   RUNG wire#w4
      Coil( "Safetyinterface".StackDoor8.monitoring.DoorLock )
   END_RUNG
   // the same network as SCL:
   "Safetyinterface".StackDoor8.monitoring.DoorOpen := #TRUE AND ("Safety.DataFromSafety".fDoorCoilStatus.stackTableRearDoorUnlock OR (NOT "Safety.DataFromSafety".fDoorCoilStatus.stackTableRearDoorUnlock AND "Safety.DataFromSafety".fDoorDrive.fDoor8.ackReq AND NOT "Global.Data".general.clock.cycle1000Msec AND NOT "Safety.DataFromSafety".fDoorSwitchStatus.stackTableRearDoorOpen));
   "Safetyinterface".StackDoor8.monitoring.DoorUnLock := #TRUE AND "Safety.DataFromSafety".fDoorCoilStatus.stackTableRearDoorUnlock;
   #_w1 := #TRUE AND NOT "Safety.DataFromSafety".fDoorCoilStatus.stackTableRearDoorUnlock AND (NOT "Safety.DataFromSafety".fDoorDrive.fDoor8.ackReq OR ("Safety.DataFromSafety".fDoorDrive.fDoor8.ackReq AND NOT "Global.Data".general.clock.cycle1000Msec));
   "Safetyinterface".StackDoor8.monitoring.DoorClose := #_w1 AND NOT "Safety.DataFromSafety".fDoorSwitchStatus.stackTableRearDoorOpen AND NOT "Safetyinterface".StackDoor8.monitoring.DoorOpen;
   "Safetyinterface".StackDoor8.monitoring.DoorLock := #_w1;
END_REGION

REGION Network 13: Stack Door Common Command#9
   RUNG wire#powerrail
      Contact( #TRUE )
      wire#w1
      Contact( "Safetyinterface".StackDoor9.commands.Lock )
      wire#w2
      Coil( "Safety.DataToSafety".StackDoor9.Lock )
   END_RUNG
   RUNG wire#w1
      P_Contact(operand := "Unit1.EmNodes".unitStatus.mode.production, bit := "TestTemp".TempBool[4])
   END_RUNG wire#w2
   RUNG wire#w1
      Contact( "Safetyinterface".StackDoor9.commands.Unlock )
      Coil( "Safety.DataToSafety".StackDoor9.Unlock )
   END_RUNG
   // the same network as SCL:
   #_w1 := #TRUE AND "Unit1.EmNodes".unitStatus.mode.production AND NOT "TestTemp".TempBool[4];   // rising edge of "Unit1.EmNodes".unitStatus.mode.production
   "TestTemp".TempBool[4] := "Unit1.EmNodes".unitStatus.mode.production;
   "Safety.DataToSafety".StackDoor9.Lock := (#TRUE AND "Safetyinterface".StackDoor9.commands.Lock) OR #_w1;
   "Safety.DataToSafety".StackDoor9.Unlock := #TRUE AND "Safetyinterface".StackDoor9.commands.Unlock;
END_REGION

REGION Network 14: Stack Door Common Monitoring#9
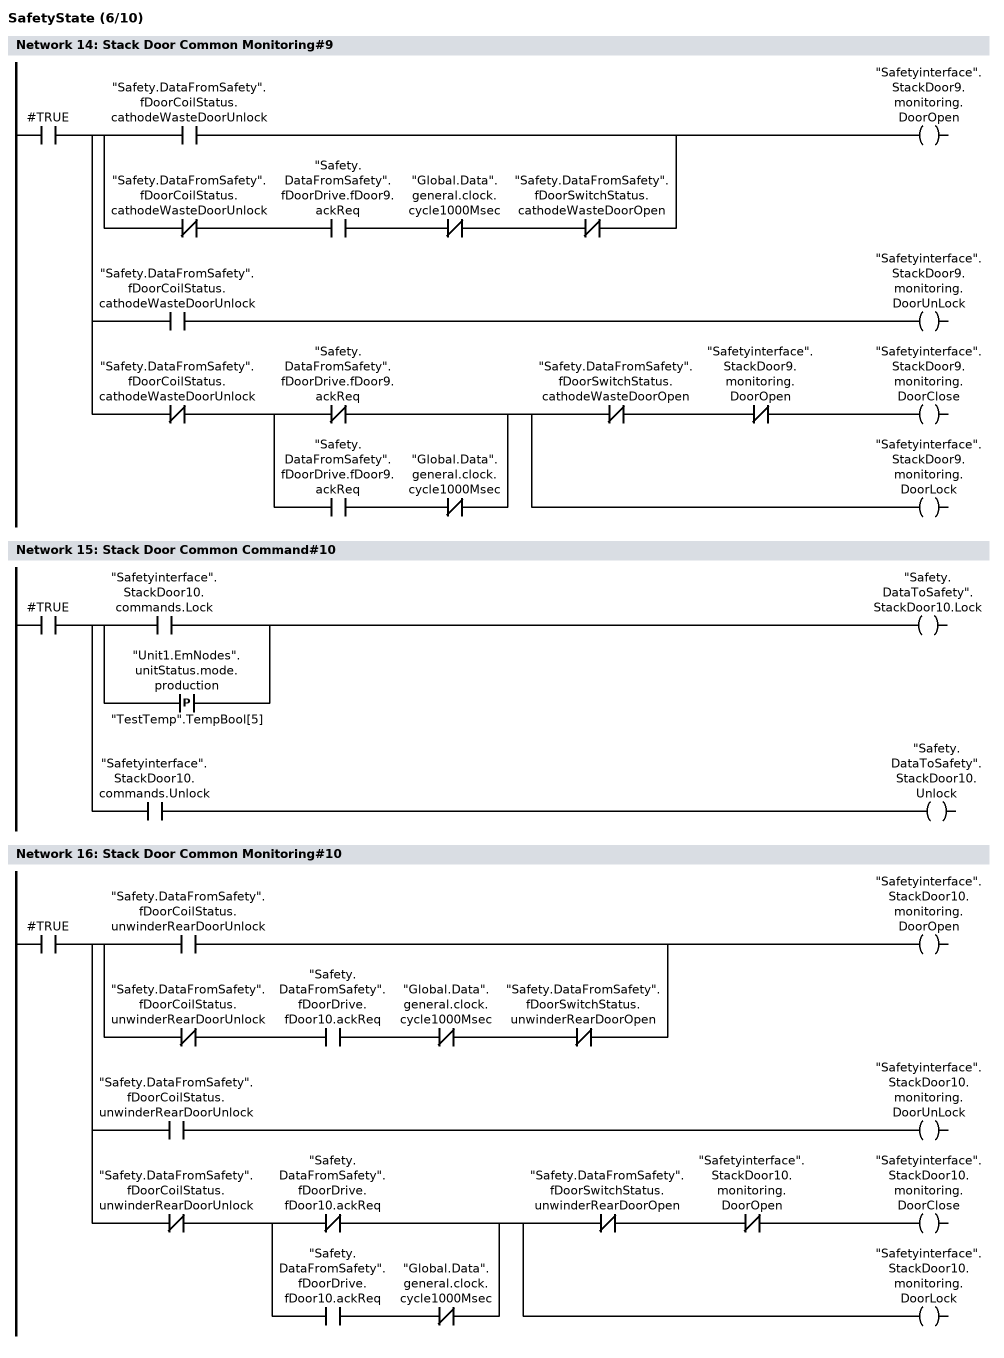
   RUNG wire#powerrail
      Contact( #TRUE )
      wire#w1
      Contact( "Safety.DataFromSafety".fDoorCoilStatus.cathodeWasteDoorUnlock )
      wire#w2
      Coil( "Safetyinterface".StackDoor9.monitoring.DoorOpen )
   END_RUNG
   RUNG wire#w1
      I_Contact( "Safety.DataFromSafety".fDoorCoilStatus.cathodeWasteDoorUnlock )
      Contact( "Safety.DataFromSafety".fDoorDrive.fDoor9.ackReq )
      I_Contact( "Global.Data".general.clock.cycle1000Msec )
      I_Contact( "Safety.DataFromSafety".fDoorSwitchStatus.cathodeWasteDoorOpen )
   END_RUNG wire#w2
   RUNG wire#w1
      Contact( "Safety.DataFromSafety".fDoorCoilStatus.cathodeWasteDoorUnlock )
      Coil( "Safetyinterface".StackDoor9.monitoring.DoorUnLock )
   END_RUNG
   RUNG wire#w1
      I_Contact( "Safety.DataFromSafety".fDoorCoilStatus.cathodeWasteDoorUnlock )
      wire#w3
      I_Contact( "Safety.DataFromSafety".fDoorDrive.fDoor9.ackReq )
      wire#w4
      I_Contact( "Safety.DataFromSafety".fDoorSwitchStatus.cathodeWasteDoorOpen )
      I_Contact( "Safetyinterface".StackDoor9.monitoring.DoorOpen )
      Coil( "Safetyinterface".StackDoor9.monitoring.DoorClose )
   END_RUNG
   RUNG wire#w3
      Contact( "Safety.DataFromSafety".fDoorDrive.fDoor9.ackReq )
      I_Contact( "Global.Data".general.clock.cycle1000Msec )
   END_RUNG wire#w4
   RUNG wire#w4
      Coil( "Safetyinterface".StackDoor9.monitoring.DoorLock )
   END_RUNG
   // the same network as SCL:
   "Safetyinterface".StackDoor9.monitoring.DoorOpen := #TRUE AND ("Safety.DataFromSafety".fDoorCoilStatus.cathodeWasteDoorUnlock OR (NOT "Safety.DataFromSafety".fDoorCoilStatus.cathodeWasteDoorUnlock AND "Safety.DataFromSafety".fDoorDrive.fDoor9.ackReq AND NOT "Global.Data".general.clock.cycle1000Msec AND NOT "Safety.DataFromSafety".fDoorSwitchStatus.cathodeWasteDoorOpen));
   "Safetyinterface".StackDoor9.monitoring.DoorUnLock := #TRUE AND "Safety.DataFromSafety".fDoorCoilStatus.cathodeWasteDoorUnlock;
   #_w1 := #TRUE AND NOT "Safety.DataFromSafety".fDoorCoilStatus.cathodeWasteDoorUnlock AND (NOT "Safety.DataFromSafety".fDoorDrive.fDoor9.ackReq OR ("Safety.DataFromSafety".fDoorDrive.fDoor9.ackReq AND NOT "Global.Data".general.clock.cycle1000Msec));
   "Safetyinterface".StackDoor9.monitoring.DoorClose := #_w1 AND NOT "Safety.DataFromSafety".fDoorSwitchStatus.cathodeWasteDoorOpen AND NOT "Safetyinterface".StackDoor9.monitoring.DoorOpen;
   "Safetyinterface".StackDoor9.monitoring.DoorLock := #_w1;
END_REGION

REGION Network 15: Stack Door Common Command#10
   RUNG wire#powerrail
      Contact( #TRUE )
      wire#w1
      Contact( "Safetyinterface".StackDoor10.commands.Lock )
      wire#w2
      Coil( "Safety.DataToSafety".StackDoor10.Lock )
   END_RUNG
   RUNG wire#w1
      P_Contact(operand := "Unit1.EmNodes".unitStatus.mode.production, bit := "TestTemp".TempBool[5])
   END_RUNG wire#w2
   RUNG wire#w1
      Contact( "Safetyinterface".StackDoor10.commands.Unlock )
      Coil( "Safety.DataToSafety".StackDoor10.Unlock )
   END_RUNG
   // the same network as SCL:
   #_w1 := #TRUE AND "Unit1.EmNodes".unitStatus.mode.production AND NOT "TestTemp".TempBool[5];   // rising edge of "Unit1.EmNodes".unitStatus.mode.production
   "TestTemp".TempBool[5] := "Unit1.EmNodes".unitStatus.mode.production;
   "Safety.DataToSafety".StackDoor10.Lock := (#TRUE AND "Safetyinterface".StackDoor10.commands.Lock) OR #_w1;
   "Safety.DataToSafety".StackDoor10.Unlock := #TRUE AND "Safetyinterface".StackDoor10.commands.Unlock;
END_REGION

REGION Network 16: Stack Door Common Monitoring#10
   RUNG wire#powerrail
      Contact( #TRUE )
      wire#w1
      Contact( "Safety.DataFromSafety".fDoorCoilStatus.unwinderRearDoorUnlock )
      wire#w2
      Coil( "Safetyinterface".StackDoor10.monitoring.DoorOpen )
   END_RUNG
   RUNG wire#w1
      I_Contact( "Safety.DataFromSafety".fDoorCoilStatus.unwinderRearDoorUnlock )
      Contact( "Safety.DataFromSafety".fDoorDrive.fDoor10.ackReq )
      I_Contact( "Global.Data".general.clock.cycle1000Msec )
      I_Contact( "Safety.DataFromSafety".fDoorSwitchStatus.unwinderRearDoorOpen )
   END_RUNG wire#w2
   RUNG wire#w1
      Contact( "Safety.DataFromSafety".fDoorCoilStatus.unwinderRearDoorUnlock )
      Coil( "Safetyinterface".StackDoor10.monitoring.DoorUnLock )
   END_RUNG
   RUNG wire#w1
      I_Contact( "Safety.DataFromSafety".fDoorCoilStatus.unwinderRearDoorUnlock )
      wire#w3
      I_Contact( "Safety.DataFromSafety".fDoorDrive.fDoor10.ackReq )
      wire#w4
      I_Contact( "Safety.DataFromSafety".fDoorSwitchStatus.unwinderRearDoorOpen )
      I_Contact( "Safetyinterface".StackDoor10.monitoring.DoorOpen )
      Coil( "Safetyinterface".StackDoor10.monitoring.DoorClose )
   END_RUNG
   RUNG wire#w3
      Contact( "Safety.DataFromSafety".fDoorDrive.fDoor10.ackReq )
      I_Contact( "Global.Data".general.clock.cycle1000Msec )
   END_RUNG wire#w4
   RUNG wire#w4
      Coil( "Safetyinterface".StackDoor10.monitoring.DoorLock )
   END_RUNG
   // the same network as SCL:
   "Safetyinterface".StackDoor10.monitoring.DoorOpen := #TRUE AND ("Safety.DataFromSafety".fDoorCoilStatus.unwinderRearDoorUnlock OR (NOT "Safety.DataFromSafety".fDoorCoilStatus.unwinderRearDoorUnlock AND "Safety.DataFromSafety".fDoorDrive.fDoor10.ackReq AND NOT "Global.Data".general.clock.cycle1000Msec AND NOT "Safety.DataFromSafety".fDoorSwitchStatus.unwinderRearDoorOpen));
   "Safetyinterface".StackDoor10.monitoring.DoorUnLock := #TRUE AND "Safety.DataFromSafety".fDoorCoilStatus.unwinderRearDoorUnlock;
   #_w1 := #TRUE AND NOT "Safety.DataFromSafety".fDoorCoilStatus.unwinderRearDoorUnlock AND (NOT "Safety.DataFromSafety".fDoorDrive.fDoor10.ackReq OR ("Safety.DataFromSafety".fDoorDrive.fDoor10.ackReq AND NOT "Global.Data".general.clock.cycle1000Msec));
   "Safetyinterface".StackDoor10.monitoring.DoorClose := #_w1 AND NOT "Safety.DataFromSafety".fDoorSwitchStatus.unwinderRearDoorOpen AND NOT "Safetyinterface".StackDoor10.monitoring.DoorOpen;
   "Safetyinterface".StackDoor10.monitoring.DoorLock := #_w1;
END_REGION

REGION Network 17: At Least One Door Unlock Command
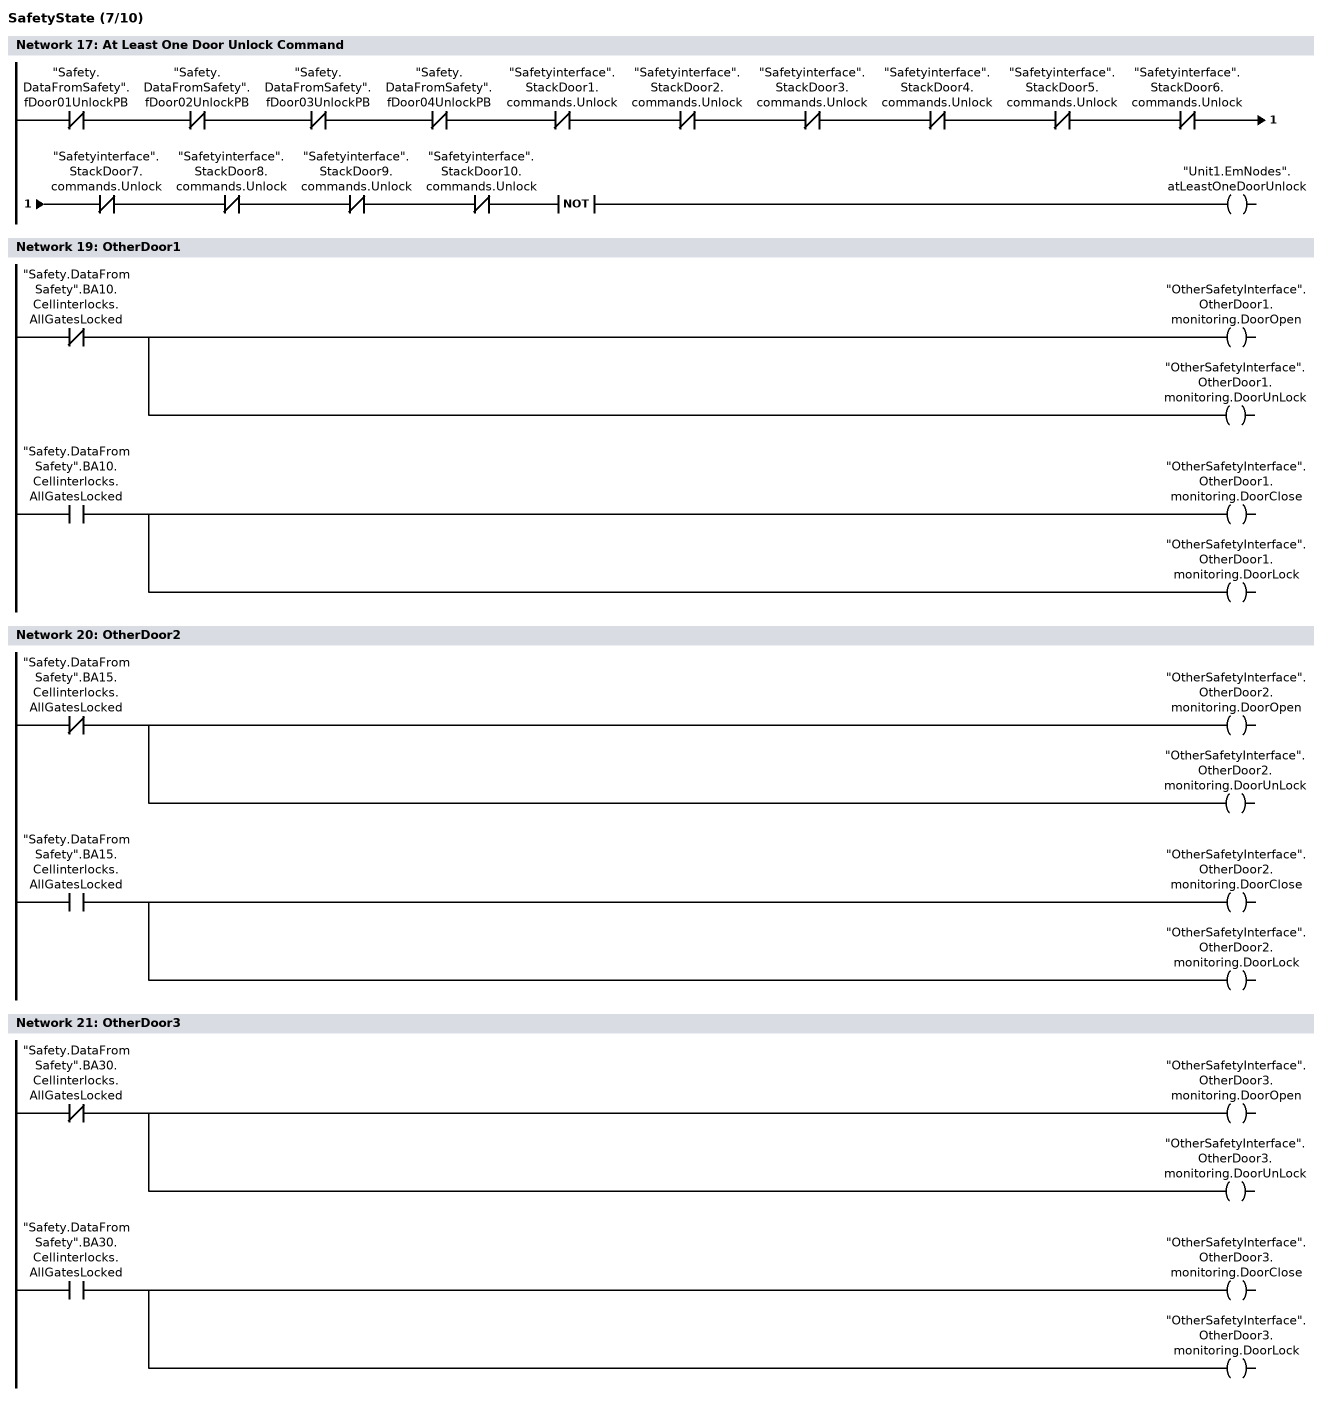
   RUNG wire#powerrail
      I_Contact( "Safety.DataFromSafety".fDoor01UnlockPB )
      I_Contact( "Safety.DataFromSafety".fDoor02UnlockPB )
      I_Contact( "Safety.DataFromSafety".fDoor03UnlockPB )
      I_Contact( "Safety.DataFromSafety".fDoor04UnlockPB )
      I_Contact( "Safetyinterface".StackDoor1.commands.Unlock )
      I_Contact( "Safetyinterface".StackDoor2.commands.Unlock )
      I_Contact( "Safetyinterface".StackDoor3.commands.Unlock )
      I_Contact( "Safetyinterface".StackDoor4.commands.Unlock )
      I_Contact( "Safetyinterface".StackDoor5.commands.Unlock )
      I_Contact( "Safetyinterface".StackDoor6.commands.Unlock )
      I_Contact( "Safetyinterface".StackDoor7.commands.Unlock )
      I_Contact( "Safetyinterface".StackDoor8.commands.Unlock )
      I_Contact( "Safetyinterface".StackDoor9.commands.Unlock )
      I_Contact( "Safetyinterface".StackDoor10.commands.Unlock )
      Not()
      Coil( "Unit1.EmNodes".atLeastOneDoorUnlock )
   END_RUNG
   // the same network as SCL:
   "Unit1.EmNodes".atLeastOneDoorUnlock := NOT (NOT "Safety.DataFromSafety".fDoor01UnlockPB AND NOT "Safety.DataFromSafety".fDoor02UnlockPB AND NOT "Safety.DataFromSafety".fDoor03UnlockPB AND NOT "Safety.DataFromSafety".fDoor04UnlockPB AND NOT "Safetyinterface".StackDoor1.commands.Unlock AND NOT "Safetyinterface".StackDoor2.commands.Unlock AND NOT "Safetyinterface".StackDoor3.commands.Unlock AND NOT "Safetyinterface".StackDoor4.commands.Unlock AND NOT "Safetyinterface".StackDoor5.commands.Unlock AND NOT "Safetyinterface".StackDoor6.commands.Unlock AND NOT "Safetyinterface".StackDoor7.commands.Unlock AND NOT "Safetyinterface".StackDoor8.commands.Unlock AND NOT "Safetyinterface".StackDoor9.commands.Unlock AND NOT "Safetyinterface".StackDoor10.commands.Unlock);
END_REGION

REGION Network 18: ***** Other Safety Interface *****
END_REGION

REGION Network 19: OtherDoor1
   RUNG wire#powerrail
      I_Contact( "Safety.DataFromSafety".BA10.Cellinterlocks.AllGatesLocked )
      wire#w1
      Coil( "OtherSafetyInterface".OtherDoor1.monitoring.DoorOpen )
   END_RUNG
   RUNG wire#w1
      Coil( "OtherSafetyInterface".OtherDoor1.monitoring.DoorUnLock )
   END_RUNG
   RUNG wire#powerrail
      Contact( "Safety.DataFromSafety".BA10.Cellinterlocks.AllGatesLocked )
      wire#w2
      Coil( "OtherSafetyInterface".OtherDoor1.monitoring.DoorClose )
   END_RUNG
   RUNG wire#w2
      Coil( "OtherSafetyInterface".OtherDoor1.monitoring.DoorLock )
   END_RUNG
   // the same network as SCL:
   "OtherSafetyInterface".OtherDoor1.monitoring.DoorOpen := NOT "Safety.DataFromSafety".BA10.Cellinterlocks.AllGatesLocked;
   "OtherSafetyInterface".OtherDoor1.monitoring.DoorUnLock := NOT "Safety.DataFromSafety".BA10.Cellinterlocks.AllGatesLocked;
   "OtherSafetyInterface".OtherDoor1.monitoring.DoorClose := "Safety.DataFromSafety".BA10.Cellinterlocks.AllGatesLocked;
   "OtherSafetyInterface".OtherDoor1.monitoring.DoorLock := "Safety.DataFromSafety".BA10.Cellinterlocks.AllGatesLocked;
END_REGION

REGION Network 20: OtherDoor2
   RUNG wire#powerrail
      I_Contact( "Safety.DataFromSafety".BA15.Cellinterlocks.AllGatesLocked )
      wire#w1
      Coil( "OtherSafetyInterface".OtherDoor2.monitoring.DoorOpen )
   END_RUNG
   RUNG wire#w1
      Coil( "OtherSafetyInterface".OtherDoor2.monitoring.DoorUnLock )
   END_RUNG
   RUNG wire#powerrail
      Contact( "Safety.DataFromSafety".BA15.Cellinterlocks.AllGatesLocked )
      wire#w2
      Coil( "OtherSafetyInterface".OtherDoor2.monitoring.DoorClose )
   END_RUNG
   RUNG wire#w2
      Coil( "OtherSafetyInterface".OtherDoor2.monitoring.DoorLock )
   END_RUNG
   // the same network as SCL:
   "OtherSafetyInterface".OtherDoor2.monitoring.DoorOpen := NOT "Safety.DataFromSafety".BA15.Cellinterlocks.AllGatesLocked;
   "OtherSafetyInterface".OtherDoor2.monitoring.DoorUnLock := NOT "Safety.DataFromSafety".BA15.Cellinterlocks.AllGatesLocked;
   "OtherSafetyInterface".OtherDoor2.monitoring.DoorClose := "Safety.DataFromSafety".BA15.Cellinterlocks.AllGatesLocked;
   "OtherSafetyInterface".OtherDoor2.monitoring.DoorLock := "Safety.DataFromSafety".BA15.Cellinterlocks.AllGatesLocked;
END_REGION

REGION Network 21: OtherDoor3
   RUNG wire#powerrail
      I_Contact( "Safety.DataFromSafety".BA30.Cellinterlocks.AllGatesLocked )
      wire#w1
      Coil( "OtherSafetyInterface".OtherDoor3.monitoring.DoorOpen )
   END_RUNG
   RUNG wire#w1
      Coil( "OtherSafetyInterface".OtherDoor3.monitoring.DoorUnLock )
   END_RUNG
   RUNG wire#powerrail
      Contact( "Safety.DataFromSafety".BA30.Cellinterlocks.AllGatesLocked )
      wire#w2
      Coil( "OtherSafetyInterface".OtherDoor3.monitoring.DoorClose )
   END_RUNG
   RUNG wire#w2
      Coil( "OtherSafetyInterface".OtherDoor3.monitoring.DoorLock )
   END_RUNG
   // the same network as SCL:
   "OtherSafetyInterface".OtherDoor3.monitoring.DoorOpen := NOT "Safety.DataFromSafety".BA30.Cellinterlocks.AllGatesLocked;
   "OtherSafetyInterface".OtherDoor3.monitoring.DoorUnLock := NOT "Safety.DataFromSafety".BA30.Cellinterlocks.AllGatesLocked;
   "OtherSafetyInterface".OtherDoor3.monitoring.DoorClose := "Safety.DataFromSafety".BA30.Cellinterlocks.AllGatesLocked;
   "OtherSafetyInterface".OtherDoor3.monitoring.DoorLock := "Safety.DataFromSafety".BA30.Cellinterlocks.AllGatesLocked;
END_REGION

REGION Network 22: OtherDoor4
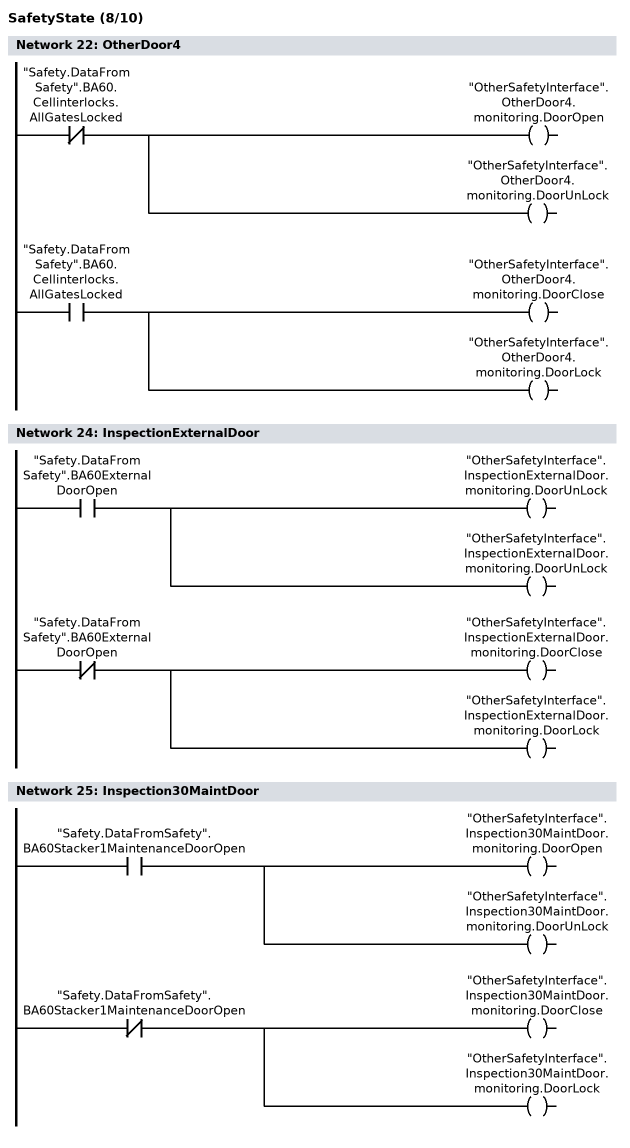
   RUNG wire#powerrail
      I_Contact( "Safety.DataFromSafety".BA60.Cellinterlocks.AllGatesLocked )
      wire#w1
      Coil( "OtherSafetyInterface".OtherDoor4.monitoring.DoorOpen )
   END_RUNG
   RUNG wire#w1
      Coil( "OtherSafetyInterface".OtherDoor4.monitoring.DoorUnLock )
   END_RUNG
   RUNG wire#powerrail
      Contact( "Safety.DataFromSafety".BA60.Cellinterlocks.AllGatesLocked )
      wire#w2
      Coil( "OtherSafetyInterface".OtherDoor4.monitoring.DoorClose )
   END_RUNG
   RUNG wire#w2
      Coil( "OtherSafetyInterface".OtherDoor4.monitoring.DoorLock )
   END_RUNG
   // the same network as SCL:
   "OtherSafetyInterface".OtherDoor4.monitoring.DoorOpen := NOT "Safety.DataFromSafety".BA60.Cellinterlocks.AllGatesLocked;
   "OtherSafetyInterface".OtherDoor4.monitoring.DoorUnLock := NOT "Safety.DataFromSafety".BA60.Cellinterlocks.AllGatesLocked;
   "OtherSafetyInterface".OtherDoor4.monitoring.DoorClose := "Safety.DataFromSafety".BA60.Cellinterlocks.AllGatesLocked;
   "OtherSafetyInterface".OtherDoor4.monitoring.DoorLock := "Safety.DataFromSafety".BA60.Cellinterlocks.AllGatesLocked;
END_REGION

REGION Network 24: InspectionExternalDoor
   RUNG wire#powerrail
      Contact( "Safety.DataFromSafety".BA60ExternalDoorOpen )
      wire#w1
      Coil( "OtherSafetyInterface".InspectionExternalDoor.monitoring.DoorUnLock )
   END_RUNG
   RUNG wire#w1
      Coil( "OtherSafetyInterface".InspectionExternalDoor.monitoring.DoorUnLock )
   END_RUNG
   RUNG wire#powerrail
      I_Contact( "Safety.DataFromSafety".BA60ExternalDoorOpen )
      wire#w2
      Coil( "OtherSafetyInterface".InspectionExternalDoor.monitoring.DoorClose )
   END_RUNG
   RUNG wire#w2
      Coil( "OtherSafetyInterface".InspectionExternalDoor.monitoring.DoorLock )
   END_RUNG
   // the same network as SCL:
   "OtherSafetyInterface".InspectionExternalDoor.monitoring.DoorUnLock := "Safety.DataFromSafety".BA60ExternalDoorOpen;
   "OtherSafetyInterface".InspectionExternalDoor.monitoring.DoorUnLock := "Safety.DataFromSafety".BA60ExternalDoorOpen;
   "OtherSafetyInterface".InspectionExternalDoor.monitoring.DoorClose := NOT "Safety.DataFromSafety".BA60ExternalDoorOpen;
   "OtherSafetyInterface".InspectionExternalDoor.monitoring.DoorLock := NOT "Safety.DataFromSafety".BA60ExternalDoorOpen;
END_REGION

REGION Network 25: Inspection30MaintDoor
   RUNG wire#powerrail
      Contact( "Safety.DataFromSafety".BA60Stacker1MaintenanceDoorOpen )
      wire#w1
      Coil( "OtherSafetyInterface".Inspection30MaintDoor.monitoring.DoorOpen )
   END_RUNG
   RUNG wire#w1
      Coil( "OtherSafetyInterface".Inspection30MaintDoor.monitoring.DoorUnLock )
   END_RUNG
   RUNG wire#powerrail
      I_Contact( "Safety.DataFromSafety".BA60Stacker1MaintenanceDoorOpen )
      wire#w2
      Coil( "OtherSafetyInterface".Inspection30MaintDoor.monitoring.DoorClose )
   END_RUNG
   RUNG wire#w2
      Coil( "OtherSafetyInterface".Inspection30MaintDoor.monitoring.DoorLock )
   END_RUNG
   // the same network as SCL:
   "OtherSafetyInterface".Inspection30MaintDoor.monitoring.DoorOpen := "Safety.DataFromSafety".BA60Stacker1MaintenanceDoorOpen;
   "OtherSafetyInterface".Inspection30MaintDoor.monitoring.DoorUnLock := "Safety.DataFromSafety".BA60Stacker1MaintenanceDoorOpen;
   "OtherSafetyInterface".Inspection30MaintDoor.monitoring.DoorClose := NOT "Safety.DataFromSafety".BA60Stacker1MaintenanceDoorOpen;
   "OtherSafetyInterface".Inspection30MaintDoor.monitoring.DoorLock := NOT "Safety.DataFromSafety".BA60Stacker1MaintenanceDoorOpen;
END_REGION

REGION Network 26: Inspection40MaintDoor
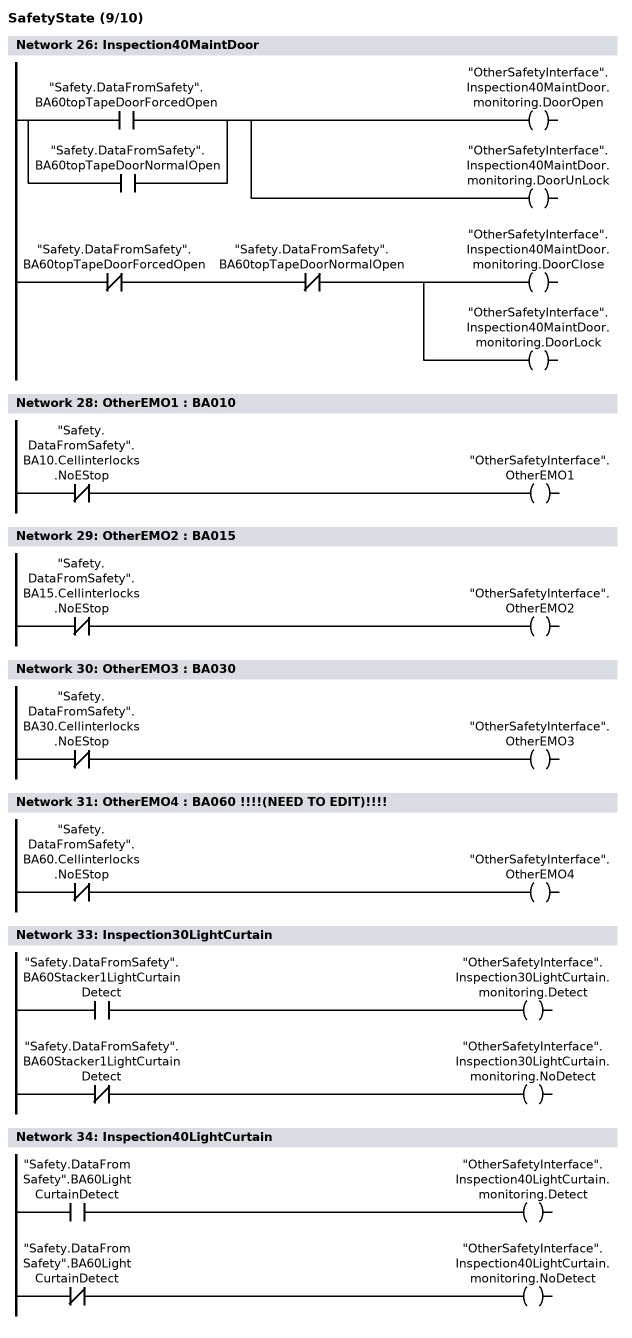
   RUNG wire#powerrail
      Contact( "Safety.DataFromSafety".BA60topTapeDoorForcedOpen )
      wire#w1
      Coil( "OtherSafetyInterface".Inspection40MaintDoor.monitoring.DoorOpen )
   END_RUNG
   RUNG wire#powerrail
      Contact( "Safety.DataFromSafety".BA60topTapeDoorNormalOpen )
   END_RUNG wire#w1
   RUNG wire#w1
      Coil( "OtherSafetyInterface".Inspection40MaintDoor.monitoring.DoorUnLock )
   END_RUNG
   RUNG wire#powerrail
      I_Contact( "Safety.DataFromSafety".BA60topTapeDoorForcedOpen )
      I_Contact( "Safety.DataFromSafety".BA60topTapeDoorNormalOpen )
      wire#w2
      Coil( "OtherSafetyInterface".Inspection40MaintDoor.monitoring.DoorClose )
   END_RUNG
   RUNG wire#w2
      Coil( "OtherSafetyInterface".Inspection40MaintDoor.monitoring.DoorLock )
   END_RUNG
   // the same network as SCL:
   "OtherSafetyInterface".Inspection40MaintDoor.monitoring.DoorOpen := "Safety.DataFromSafety".BA60topTapeDoorForcedOpen OR "Safety.DataFromSafety".BA60topTapeDoorNormalOpen;
   "OtherSafetyInterface".Inspection40MaintDoor.monitoring.DoorUnLock := "OtherSafetyInterface".Inspection40MaintDoor.monitoring.DoorOpen;
   "OtherSafetyInterface".Inspection40MaintDoor.monitoring.DoorClose := NOT "Safety.DataFromSafety".BA60topTapeDoorForcedOpen AND NOT "Safety.DataFromSafety".BA60topTapeDoorNormalOpen;
   "OtherSafetyInterface".Inspection40MaintDoor.monitoring.DoorLock := "OtherSafetyInterface".Inspection40MaintDoor.monitoring.DoorClose;
END_REGION

REGION Network 28: OtherEMO1 : BA010
   RUNG wire#powerrail
      I_Contact( "Safety.DataFromSafety".BA10.Cellinterlocks.NoEStop )
      Coil( "OtherSafetyInterface".OtherEMO1 )
   END_RUNG
   // the same network as SCL:
   "OtherSafetyInterface".OtherEMO1 := NOT "Safety.DataFromSafety".BA10.Cellinterlocks.NoEStop;
END_REGION

REGION Network 29: OtherEMO2 : BA015
   RUNG wire#powerrail
      I_Contact( "Safety.DataFromSafety".BA15.Cellinterlocks.NoEStop )
      Coil( "OtherSafetyInterface".OtherEMO2 )
   END_RUNG
   // the same network as SCL:
   "OtherSafetyInterface".OtherEMO2 := NOT "Safety.DataFromSafety".BA15.Cellinterlocks.NoEStop;
END_REGION

REGION Network 30: OtherEMO3 : BA030
   RUNG wire#powerrail
      I_Contact( "Safety.DataFromSafety".BA30.Cellinterlocks.NoEStop )
      Coil( "OtherSafetyInterface".OtherEMO3 )
   END_RUNG
   // the same network as SCL:
   "OtherSafetyInterface".OtherEMO3 := NOT "Safety.DataFromSafety".BA30.Cellinterlocks.NoEStop;
END_REGION

REGION Network 31: OtherEMO4 : BA060 !!!!(NEED TO EDIT)!!!!
   RUNG wire#powerrail
      I_Contact( "Safety.DataFromSafety".BA60.Cellinterlocks.NoEStop )
      Coil( "OtherSafetyInterface".OtherEMO4 )
   END_RUNG
   // the same network as SCL:
   "OtherSafetyInterface".OtherEMO4 := NOT "Safety.DataFromSafety".BA60.Cellinterlocks.NoEStop;
END_REGION

REGION Network 33: Inspection30LightCurtain
   RUNG wire#powerrail
      Contact( "Safety.DataFromSafety".BA60Stacker1LightCurtainDetect )
      Coil( "OtherSafetyInterface".Inspection30LightCurtain.monitoring.Detect )
   END_RUNG
   RUNG wire#powerrail
      I_Contact( "Safety.DataFromSafety".BA60Stacker1LightCurtainDetect )
      Coil( "OtherSafetyInterface".Inspection30LightCurtain.monitoring.NoDetect )
   END_RUNG
   // the same network as SCL:
   "OtherSafetyInterface".Inspection30LightCurtain.monitoring.Detect := "Safety.DataFromSafety".BA60Stacker1LightCurtainDetect;
   "OtherSafetyInterface".Inspection30LightCurtain.monitoring.NoDetect := NOT "Safety.DataFromSafety".BA60Stacker1LightCurtainDetect;
END_REGION

REGION Network 34: Inspection40LightCurtain
   RUNG wire#powerrail
      Contact( "Safety.DataFromSafety".BA60LightCurtainDetect )
      Coil( "OtherSafetyInterface".Inspection40LightCurtain.monitoring.Detect )
   END_RUNG
   RUNG wire#powerrail
      I_Contact( "Safety.DataFromSafety".BA60LightCurtainDetect )
      Coil( "OtherSafetyInterface".Inspection40LightCurtain.monitoring.NoDetect )
   END_RUNG
   // the same network as SCL:
   "OtherSafetyInterface".Inspection40LightCurtain.monitoring.Detect := "Safety.DataFromSafety".BA60LightCurtainDetect;
   "OtherSafetyInterface".Inspection40LightCurtain.monitoring.NoDetect := NOT "Safety.DataFromSafety".BA60LightCurtainDetect;
END_REGION

REGION Network 36: 30CathodeConveyorCover
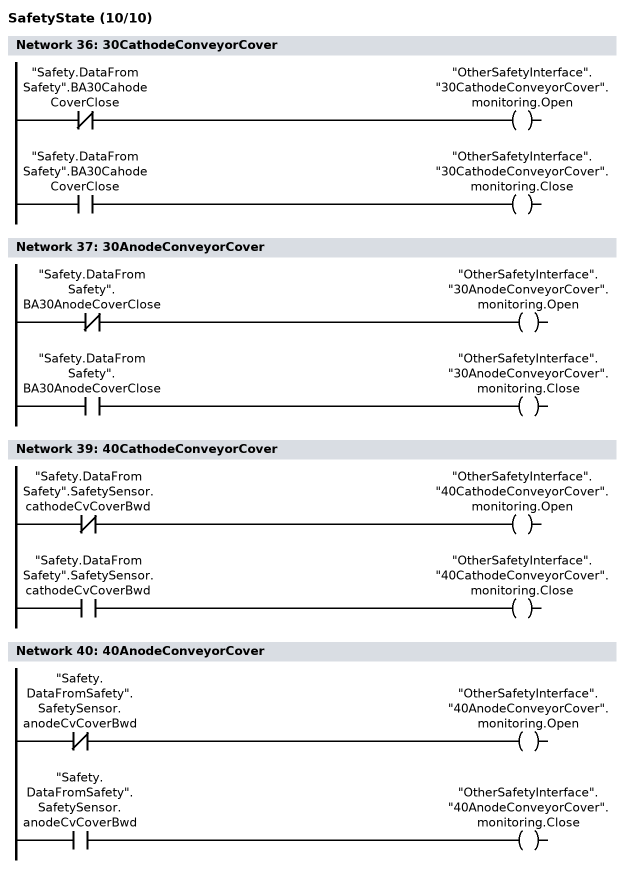
   RUNG wire#powerrail
      I_Contact( "Safety.DataFromSafety".BA30CahodeCoverClose )
      Coil( "OtherSafetyInterface"."30CathodeConveyorCover".monitoring.Open )
   END_RUNG
   RUNG wire#powerrail
      Contact( "Safety.DataFromSafety".BA30CahodeCoverClose )
      Coil( "OtherSafetyInterface"."30CathodeConveyorCover".monitoring.Close )
   END_RUNG
   // the same network as SCL:
   "OtherSafetyInterface"."30CathodeConveyorCover".monitoring.Open := NOT "Safety.DataFromSafety".BA30CahodeCoverClose;
   "OtherSafetyInterface"."30CathodeConveyorCover".monitoring.Close := "Safety.DataFromSafety".BA30CahodeCoverClose;
END_REGION

REGION Network 37: 30AnodeConveyorCover
   RUNG wire#powerrail
      I_Contact( "Safety.DataFromSafety".BA30AnodeCoverClose )
      Coil( "OtherSafetyInterface"."30AnodeConveyorCover".monitoring.Open )
   END_RUNG
   RUNG wire#powerrail
      Contact( "Safety.DataFromSafety".BA30AnodeCoverClose )
      Coil( "OtherSafetyInterface"."30AnodeConveyorCover".monitoring.Close )
   END_RUNG
   // the same network as SCL:
   "OtherSafetyInterface"."30AnodeConveyorCover".monitoring.Open := NOT "Safety.DataFromSafety".BA30AnodeCoverClose;
   "OtherSafetyInterface"."30AnodeConveyorCover".monitoring.Close := "Safety.DataFromSafety".BA30AnodeCoverClose;
END_REGION

REGION Network 39: 40CathodeConveyorCover
   RUNG wire#powerrail
      I_Contact( "Safety.DataFromSafety".SafetySensor.cathodeCvCoverBwd )
      Coil( "OtherSafetyInterface"."40CathodeConveyorCover".monitoring.Open )
   END_RUNG
   RUNG wire#powerrail
      Contact( "Safety.DataFromSafety".SafetySensor.cathodeCvCoverBwd )
      Coil( "OtherSafetyInterface"."40CathodeConveyorCover".monitoring.Close )
   END_RUNG
   // the same network as SCL:
   "OtherSafetyInterface"."40CathodeConveyorCover".monitoring.Open := NOT "Safety.DataFromSafety".SafetySensor.cathodeCvCoverBwd;
   "OtherSafetyInterface"."40CathodeConveyorCover".monitoring.Close := "Safety.DataFromSafety".SafetySensor.cathodeCvCoverBwd;
END_REGION

REGION Network 40: 40AnodeConveyorCover
   RUNG wire#powerrail
      I_Contact( "Safety.DataFromSafety".SafetySensor.anodeCvCoverBwd )
      Coil( "OtherSafetyInterface"."40AnodeConveyorCover".monitoring.Open )
   END_RUNG
   RUNG wire#powerrail
      Contact( "Safety.DataFromSafety".SafetySensor.anodeCvCoverBwd )
      Coil( "OtherSafetyInterface"."40AnodeConveyorCover".monitoring.Close )
   END_RUNG
   // the same network as SCL:
   "OtherSafetyInterface"."40AnodeConveyorCover".monitoring.Open := NOT "Safety.DataFromSafety".SafetySensor.anodeCvCoverBwd;
   "OtherSafetyInterface"."40AnodeConveyorCover".monitoring.Close := "Safety.DataFromSafety".SafetySensor.anodeCvCoverBwd;
END_REGION
END_FUNCTION
